PROGRAM P_Demo_F_BA_UDIVal
VAR
    argNValue                      : BOOL                           := FALSE; // nValue
    fnReturn                       : U_BA_ClassValue; // 返回值
END_VAR

// =============================================================================
// Tc3_BA2_Common.F_BA_UDIVal 演示程序
// =============================================================================
// 场景：累计能耗（UDINT 千瓦时）、累计运行小时数等"非负大数"类型测点统一上报。
//
// 价值：同其它 ClassValue 系列。
//
// 验证：登录 PLC 后，按例程内变量在线写值；监视输出 / 返回值，结合 §1 功能
//       简述的预期行为对照（详见配套 .md 文档 §7 业务场景）。
//
// 验证步骤：
//   1. 右键 PLC 项目下 POUs 文件夹 → Add → Existing Item → 选本 .TcPOU 文件
//   2. 引用 Tc3_BA2_Common（References → Add library）
//   3. 编译 → 登录 → 运行；按上方『验证』指引在线写值观察
// =============================================================================

fnReturn := F_BA_UDIVal(
    nValue                   := argNValue
);

END_PROGRAM

(* stored: Version 1.1.0.1, ProductVersion 3.1.4024.5
   POU P_Demo_F_BA_UDIVal: Id {573e7a60-895b-5954-b267-a18ad9812551}, SpecialFunc None *)
